FUNCTION_BLOCK FB_ExtBase EXTENDS FB_Base
VAR_INPUT
END_VAR
VAR_OUTPUT
END_VAR
VAR
END_VAR

{attribute 'monitoring' := 'call'}
PROPERTY CalcCounter : INT
GET
END_GET
END_PROPERTY

{attribute 'TcRpcEnable'}
METHOD ResetCalcCounter : BOOL
VAR_INPUT
END_VAR
_CalcCounter := 0;
END_METHOD

END_FUNCTION_BLOCK

(* stored: Version 1.1.0.1, ProductVersion 3.1.4024.4
   POU FB_ExtBase: Id {1ab1edfc-eaca-4163-a3d9-89b9003bda36}, SpecialFunc None
   Property CalcCounter: Id {e25c9eb2-8a79-4b2f-aa7c-0e57f7945920}
   Get Get: Id {06227bd2-54ef-4a3a-b5bf-6e46c72afd9b}
   Method ResetCalcCounter: Id {b2279c0b-5c7a-4983-a2f2-267a91ab785e} *)
